// TIA Portal V16 export
// export: Created 2022-02-19T12:47:23.5808438Z, ExportSetting WithDefaults, DisplayName Totally Integrated Automation Portal, DisplayVersion V16 Update 5, DisplayName TIA Portal Version Control Interface, DisplayVersion V16 Update 2, DisplayName TIA Portal Openness, DisplayVersion V16 Update 5, DisplayName STEP 7 Professional, DisplayVersion V16 Update 5, DisplayName STEP 7 Safety, DisplayVersion V16, DisplayName WinCC Professional, DisplayVersion V16 Update 5
VAR_GLOBAL   // PLC tag table "Tabla de variables estándar"
   S0 AT %I0.0 : Bool;
   S1 AT %I0.1 : Bool;
   S2 AT %I0.2 : Bool;
   S3 AT %I0.3 : Bool;
   S4 AT %I0.4 : Bool;
   S5 AT %I0.5 : Bool;
   S6 AT %I0.6 : Bool;
   S7 AT %I0.7 : Bool;
   S8 AT %I1.0 : Bool;
   S9 AT %I1.1 : Bool;
   S10 AT %I1.2 : Bool;
   S11 AT %I1.3 : Bool;
   S12 AT %I1.4 : Bool;
   S13 AT %I1.5 : Bool;
   Y0 AT %Q0.0 : Bool;
   Y1 AT %Q0.1 : Bool;
   Y2 AT %Q0.2 : Bool;
   Y3 AT %Q0.3 : Bool;
   Y4 AT %Q0.4 : Bool;
   Y5 AT %Q0.5 : Bool;
   Y6 AT %Q0.6 : Bool;
   Y7 AT %Q0.7 : Bool;
   Y8 AT %Q1.0 : Bool;
   Y9 AT %Q1.1 : Bool;
   B0 AT %I2.0 : Bool;
   B1 AT %I2.1 : Bool;
   B2 AT %I2.2 : Bool;
   B3 AT %I2.3 : Bool;
   B4 AT %I2.4 : Bool;
   B5 AT %I2.5 : Bool;
   B6 AT %I2.6 : Bool;
   B7 AT %I2.7 : Bool;
   B8 AT %I3.0 : Bool;
   B9 AT %I3.1 : Bool;
   B10 AT %I3.2 : Bool;
   B11 AT %I3.3 : Bool;
   B12 AT %I3.4 : Bool;
   B13 AT %I3.5 : Bool;
   B14 AT %I3.6 : Bool;
   B15 AT %I3.7 : Bool;
   KM0 AT %Q2.0 : Bool;
   KM1 AT %Q2.1 : Bool;
   KM2 AT %Q2.2 : Bool;
   KM3 AT %Q2.3 : Bool;
   KM4 AT %Q2.4 : Bool;
   KM5 AT %Q2.5 : Bool;
   KM6 AT %Q2.6 : Bool;
   KM7 AT %Q2.7 : Bool;
   KM8 AT %Q3.0 : Bool;
   KM9 AT %Q3.1 : Bool;
   KM10 AT %Q3.2 : Bool;
   KM11 AT %Q3.3 : Bool;
   KM12 AT %Q3.4 : Bool;
   KM13 AT %Q3.5 : Bool;
   KM14 AT %Q3.6 : Bool;
   KM15 AT %Q3.7 : Bool;
END_VAR
